PROGRAM prgMain
VAR
	fb_Reboot		: NT_reboot;
	m_Reboot		: BOOL:=FALSE;
END_VAR

fb_Reboot(	netid := '',
			delay := 2,
			start := m_Reboot);

END_PROGRAM

(* stored: Version 1.1.0.1, ProductVersion 3.1.4024.11
   POU prgMain: Id {d730d8b7-7417-4985-b08a-48cca9bed062}, SpecialFunc None *)
